// TIA Portal V17 export
// export: Created 2024-08-20T11:55:54.4278422Z, ExportSetting WithDefaults, DisplayName Totally Integrated Automation Portal, DisplayVersion V17 Update 4, DisplayName TIA Portal Openness, DisplayVersion V17 Update 4, DisplayName TIA Portal Version Control Interface, DisplayVersion V17, DisplayName STEP 7 Professional, DisplayVersion V17 Update 4, DisplayName STEP 7 Safety, DisplayVersion V17, DisplayName WinCC Advanced, DisplayVersion V17 Update 4
DATA_BLOCK "teste_DB"   // DB6
VERSION : 0.1
// stored: AutoNumber true, DBAccessibleFromOPCUA true, InstanceOfName teste, InstanceOfType FB
"teste"
   // VAR
   //    tag1 : Int;
   //    tag2 : Int;
   //    tag3 : Int;
   // END_VAR
BEGIN
END_DATA_BLOCK
